FUNCTION_BLOCK F_ROL (* rotate left *)
  (* Standard: 61131-3; Classification: standard bit shift function *)
  (* Version 0.0, 2013-04-14, 4DIAC-IDE, 4DIAC-Consortium *)
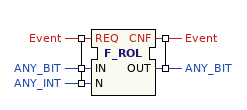
  EVENT_INPUT
    REQ WITH IN, N; (* Service Request *)
  END_EVENT
  EVENT_OUTPUT
    CNF WITH OUT; (* Confirmation of Requested Service *)
  END_EVENT
  VAR_INPUT
    IN : ANY_BIT; (* left-rotated *)
    N : ANY_INT; (* left-rotated by N bits *)
  END_VAR
  VAR_OUTPUT
    OUT : ANY_BIT; (* left-rotated by N zero-filled on right *)
  END_VAR
END_FUNCTION_BLOCK
